# EPICS substitutions: motorSimApp/iocsh/EXAMPLE_motorSim8x.substitutions
file "$(MOTOR)/db/asyn_motor.db"
{
pattern
{N,  M,        ADDR,  DESC,          EGU,      DIR,  VELO,  VBAS,  ACCL,  BDST,  BVEL,  BACC,  MRES,  PREC,  INIT}
{1,  "m$(N)",  0,     "motor $(N)",  degrees,  Pos,  1,     .1,    .2,    0,     1,     .2,    0.01,  5,     ""}
{2,  "m$(N)",  1,     "motor $(N)",  degrees,  Pos,  1,     .1,    .2,    0,     1,     .2,    0.01,  5,     ""}
{3,  "m$(N)",  2,     "motor $(N)",  degrees,  Pos,  1,     .1,    .2,    0,     1,     .2,    0.01,  5,     ""}
{4,  "m$(N)",  3,     "motor $(N)",  degrees,  Pos,  1,     .1,    .2,    0,     1,     .2,    0.01,  5,     ""}
{5,  "m$(N)",  4,     "motor $(N)",  degrees,  Pos,  1,     .1,    .2,    0,     1,     .2,    0.01,  5,     ""}
{6,  "m$(N)",  5,     "motor $(N)",  degrees,  Pos,  1,     .1,    .2,    0,     1,     .2,    0.01,  5,     ""}
{7,  "m$(N)",  6,     "motor $(N)",  degrees,  Pos,  1,     .1,    .2,    0,     1,     .2,    0.01,  5,     ""}
{8,  "m$(N)",  7,     "motor $(N)",  degrees,  Pos,  1,     .1,    .2,    0,     1,     .2,    0.01,  5,     ""}
}
